(* PLC project tennessee-eastman-chemical, Generated TextualNotationConverter 1.0 *)
(* stored: creationDateTime 2025-07-30T12:00:00, modificationDateTime 2025-01-30T12:00:00 *)

FUNCTION_BLOCK ANALOG_IN
  VAR_INPUT
    Name : STRING;
    Description : STRING;
    Raw_Signal : REAL;
    PV_High : REAL;
    PV_Low : REAL;
    Scaling_Slope : REAL;
    Scaling_Offset : REAL;
    Alarm_Enable : BOOL;
  END_VAR
  VAR_OUTPUT
    PV : REAL;
    High_Alarm : BOOL;
    Low_Alarm : BOOL;
    General_Fault : BOOL;
  END_VAR

            
          
END_FUNCTION_BLOCK

FUNCTION_BLOCK BOOL_IN
  VAR_INPUT
    Name : STRING;
    Description : STRING;
    Bool_In : BOOL;
    Alarm_OnTrue : BOOL;
    Alarm_OnFalse : BOOL;
    Latch_Enable : BOOL;
    Reset_Latch : BOOL;
  END_VAR
  VAR_OUTPUT
    Bool_Out : BOOL;
    Alarm_Active : BOOL;
    Latched_Status : BOOL;
  END_VAR

            
          
END_FUNCTION_BLOCK

FUNCTION_BLOCK DIGITAL_IN
  VAR_INPUT
    Name : STRING;
    Description : STRING;
    DI_Raw : BOOL;
    DebounceTime : STRING;
    EnableAlarm : BOOL;
  END_VAR
  VAR_OUTPUT
    DI_Out : BOOL;
    Fault_State : BOOL;
  END_VAR

            
          
END_FUNCTION_BLOCK

FUNCTION_BLOCK PID_BASIC
  VAR_INPUT
    Name : STRING;
    Description : STRING;
    AUTO : BOOL;
    PV : REAL;
    SP : REAL;
    MV_MIN : REAL;
    MV_MAX : REAL;
    X0 : REAL;
    KP : REAL;
    TR : REAL;
    TD : REAL;
    PV_High : REAL;
    PV_Low : REAL;
    Deviation_Limit : REAL;
    Inhibit : BOOL;
  END_VAR
  VAR_OUTPUT
    PV_High_Alarm : BOOL;
    PV_Low_Alarm : BOOL;
    Deviation_Alarm : BOOL;
    XOUT : REAL;
  END_VAR

            
          
END_FUNCTION_BLOCK

FUNCTION_BLOCK VALVE_ELECTRIC
  VAR_INPUT
    Name : STRING;
    Description : STRING;
    Control_Signal : REAL;
    Manual_Mode : BOOL;
    Manual_Position : REAL;
    Open_Limit : REAL;
    Close_Limit : REAL;
    Timeout : STRING;
    Inhibit : BOOL;
  END_VAR
  VAR_OUTPUT
    Valve_Position : REAL;
    Feedback_Pos : REAL;
    Valve_Moving : BOOL;
    Position_Error : BOOL;
    Alarm : BOOL;
  END_VAR

            
          
END_FUNCTION_BLOCK

FUNCTION_BLOCK VALVE_ON_OFF
  VAR_INPUT
    Name : STRING;
    Description : STRING;
    Open_Cmd : BOOL;
    Close_Cmd : BOOL;
    Timeout : STRING;
    Inhibit : BOOL;
  END_VAR
  VAR_OUTPUT
    FB_Opened : BOOL;
    FB_Closed : BOOL;
    Valve_Open_Out : BOOL;
    Valve_Close_Out : BOOL;
    Alarm_Position_Error : BOOL;
    Alarm_General : BOOL;
  END_VAR

            
          
END_FUNCTION_BLOCK

PROGRAM Section2
  VAR
    FIT_101_Raw_mA : REAL;
    FIT_101_FlowRate_GPM : REAL;
    FIC_104_MV_Percent : REAL;
    PV_103_Feedback_Position_Percent : REAL;
    PI_001_Raw_mA : REAL;
    PI_001_Pressure_psig : REAL;
  END_VAR
  VAR
    FIT-101 : ANALOG_IN;
    FIC-104 : PID_BASIC;
    PV-103 : VALVE_ELECTRIC;
    XV-106 : VALVE_ON_OFF;
    PI-001 : ANALOG_IN;
    IAL-101 : BOOL_IN;
    FAL-101 : DIGITAL_IN;
    FAL-102 : DIGITAL_IN;
    FAL-103 : DIGITAL_IN;
  END_VAR
  VAR  (* added by the conversion: wires and edge detectors of the diagram *)
    _OR2_OUT : BOOL;
  END_VAR

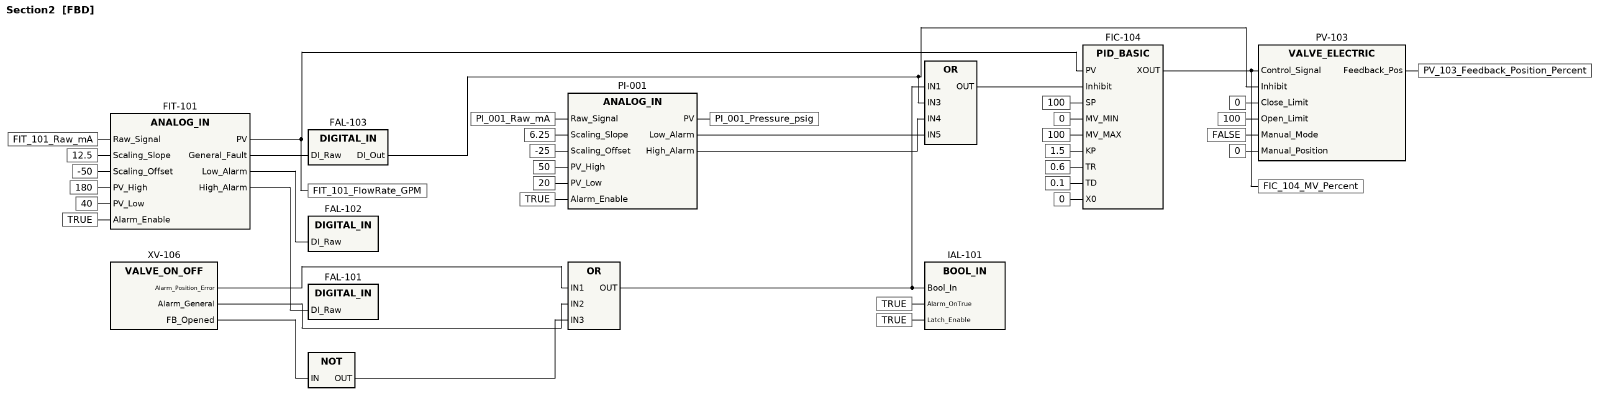
(* FBD diagram, written out as Structured Text *)
FIT-101(Raw_Signal := FIT_101_Raw_mA, Scaling_Slope := 12.5, Scaling_Offset := -50, PV_High := 180, PV_Low := 40, Alarm_Enable := TRUE);
XV-106();
_OR2_OUT := XV-106.Alarm_Position_Error OR XV-106.Alarm_General OR NOT XV-106.FB_Opened;
FAL-103(DI_Raw := FIT-101.General_Fault);
PI-001(Raw_Signal := PI_001_Raw_mA, Scaling_Slope := 6.25, Scaling_Offset := -25, PV_High := 50, PV_Low := 20, Alarm_Enable := TRUE);
FIC-104(PV := FIT-101.PV, Inhibit := _OR2_OUT OR FAL-103.DI_Out OR PI-001.High_Alarm OR PI-001.Low_Alarm, SP := 100, MV_MIN := 0, MV_MAX := 100, KP := 1.5, TR := 0.6, TD := 0.1, X0 := 0);
FIC_104_MV_Percent := FIC-104.XOUT;
FIT_101_FlowRate_GPM := FIT-101.PV;
PI_001_Pressure_psig := PI-001.PV;
PV-103(Control_Signal := FIC-104.XOUT, Inhibit := FAL-103.DI_Out, Close_Limit := 0, Open_Limit := 100, Manual_Mode := FALSE, Manual_Position := 0);
PV_103_Feedback_Position_Percent := PV-103.Feedback_Pos;
IAL-101(Bool_In := _OR2_OUT, Alarm_OnTrue := TRUE, Latch_Enable := TRUE);
FAL-101(DI_Raw := FIT-101.High_Alarm);
FAL-102(DI_Raw := FIT-101.Low_Alarm);
END_PROGRAM

FUNCTION_BLOCK DUTY_STANDBY
  VAR_INPUT
    Name : STRING;
    Description : STRING;
    Enable : BOOL;
    StartRequest : BOOL;
    AlternateEnable : BOOL;
    ForcePumpA : BOOL;
    ForcePumpB : BOOL;
    DutyElapsed : BOOL;
    MinRunElapsed : BOOL;
    SwitchoverDelayElapsed : BOOL;
    StartTimeoutElapsed : BOOL;
    PumpA_RunFB : BOOL;
    PumpB_RunFB : BOOL;
    PumpA_Fault : BOOL;
    PumpB_Fault : BOOL;
    Reset : BOOL;
    Inhibit : BOOL;
  END_VAR
  VAR_OUTPUT
    CmdPumpA : BOOL;
    CmdPumpB : BOOL;
    ActiveIsA : BOOL;
    SwitchedDueToDuty : BOOL;
    SwitchedDueToFailure : BOOL;
    Alarm_FailedStart_A : BOOL;
    Alarm_FailedStart_B : BOOL;
    Alarm_NoAvailablePump : BOOL;
  END_VAR

            
          
END_FUNCTION_BLOCK

FUNCTION_BLOCK MOTOR_2SPD
  VAR_INPUT
    Name : STRING;
    Description : STRING;
    Start_Cmd : BOOL;
    Stop_Cmd : BOOL;
    Speed_High_Cmd : BOOL;
    Speed_Low_Cmd : BOOL;
    Inhibit : BOOL;
  END_VAR
  VAR_OUTPUT
    Motor_Start_Out : BOOL;
    FB_Running : BOOL;
    FB_Trip : BOOL;
    FB_HighSpeed : BOOL;
    FB_LowSpeed : BOOL;
    Alarm_Speed_Error : BOOL;
  END_VAR

            
          
END_FUNCTION_BLOCK

FUNCTION_BLOCK MOTOR_ON_OFF
  VAR_INPUT
    Name : STRING;
    Description : STRING;
    Start_Cmd : BOOL;
    Stop_Cmd : BOOL;
    Start_Delay : STRING;
    MinRunTime : STRING;
    Inhibit : BOOL;
  END_VAR
  VAR_OUTPUT
    Motor_Start_Out : BOOL;
    FB_Running : BOOL;
    FB_Trip : BOOL;
    Alarm_Start_Fail : BOOL;
    Alarm_Stop_Fail : BOOL;
  END_VAR

            
          
END_FUNCTION_BLOCK

FUNCTION_BLOCK MOTOR_VSD
  VAR_INPUT
    Name : STRING;
    Description : STRING;
    Start_Cmd : BOOL;
    Stop_Cmd : BOOL;
    Speed_SP : REAL;
    Accel_Ramp : STRING;
    Decel_Ramp : STRING;
    Inhibit : BOOL;
  END_VAR
  VAR_OUTPUT
    Speed_Out : REAL;
    FB_Running : BOOL;
    FB_Fault : BOOL;
    FB_Ready : BOOL;
    FB_ActualSpeed : REAL;
    Alarm_Speed_Deviation : BOOL;
    Alarm_Comm_Fail : BOOL;
  END_VAR

            
          
END_FUNCTION_BLOCK

FUNCTION_BLOCK RATIO_CONTROL
  VAR_INPUT
    Name : STRING;
    Description : STRING;
    Auto : BOOL;
    PrimaryPV : REAL;
    SecondaryPV : REAL;
    RatioSP : REAL;
    Bias : REAL;
    TrimKp : REAL;
    TrimTi : STRING;
    MV_MIN : REAL;
    MV_MAX : REAL;
    ManOut : REAL;
    Inhibit : BOOL;
  END_VAR
  VAR_OUTPUT
    SlaveSP : REAL;
    ActiveRatio : REAL;
    RatioErr : REAL;
  END_VAR

            
          
END_FUNCTION_BLOCK

FUNCTION_BLOCK SPLIT_RANGE
  VAR_INPUT
    Name : STRING;
    Description : STRING;
    IN : REAL;
    Split_Point : REAL;
    Output1_Start : REAL;
    Output1_End : REAL;
    Output2_Start : REAL;
    Output2_End : REAL;
  END_VAR
  VAR_OUTPUT
    OUT1 : REAL;
    OUT2 : REAL;
  END_VAR

            
          
END_FUNCTION_BLOCK

FUNCTION_BLOCK VOTING_ANALOG
  VAR_INPUT
    Name : STRING;
    Description : STRING;
    Input1 : REAL;
    Input2 : REAL;
    Input3 : REAL;
    Deviation_Limit : REAL;
    Voting_Scheme : STRING;
    EnableAlarm : BOOL;
    Inhibit : BOOL;
  END_VAR
  VAR_OUTPUT
    Voted_Output : REAL;
    Sensor1_Fault : BOOL;
    Sensor2_Fault : BOOL;
    Sensor3_Fault : BOOL;
    Alarm_Voting_Error : BOOL;
    Healthy_Sensors_Count : INT;
  END_VAR

            
          
END_FUNCTION_BLOCK

PROGRAM Section3
  VAR
    TIT103_PV_Temperature : REAL;
    LT105_Level_PV : REAL;
    TIC101_MV_to_XV102 : REAL;
    LIC106_MV_to_LV104 : REAL;
  END_VAR
  VAR
    TIT-103 : ANALOG_IN;
    LT-105 : ANALOG_IN;
    FC-004 : ANALOG_IN;
    TIC-101 : PID_BASIC;
    LIC-106 : PID_BASIC;
    XV-102 : VALVE_ELECTRIC;
    LV-104 : VALVE_ELECTRIC;
  END_VAR

(* FBD diagram, written out as Structured Text *)
LT-105(PV_High := 80.0, PV_Low := 20.0, Alarm_Enable := TRUE, Scaling_Slope := 6.25, Scaling_Offset := -25.0);
LV-104(Control_Signal := LIC-106.XOUT, Inhibit := LT-105.High_Alarm, Manual_Mode := LT-105.High_Alarm, Open_Limit := 100.0, Close_Limit := 0.0, Manual_Position := 0.0);
TIT-103(PV_High := 200.0, PV_Low := 160.0, Alarm_Enable := TRUE, Scaling_Slope := 15.625, Scaling_Offset := -62.5);
FC-004(PV_Low := 10.0, Alarm_Enable := TRUE);
TIC-101(PV := TIT-103.PV, Inhibit := XV-102.Position_Error OR TIT-103.High_Alarm OR FC-004.Low_Alarm OR TIT-103.General_Fault, AUTO := TON(FC-004.PV > 10.0, T#21s) AND NOT XV-102.Position_Error, SP := 180.0, MV_MIN := 0.0, MV_MAX := 100.0, KP := 3.0, TR := 1.2, TD := 0.1, PV_High := 200.0, PV_Low := 160.0);
XV-102(Control_Signal := TIC-101.XOUT, Inhibit := TIT-103.High_Alarm, Manual_Mode := TIT-103.High_Alarm, Open_Limit := 100.0, Close_Limit := 0.0, Timeout := T#5s, Manual_Position := 0.0);
LIC-106(PV := LT-105.PV, Inhibit := LV-104.Position_Error OR LT-105.General_Fault OR XV-102.Alarm, AUTO := NOT XV-102.Alarm AND TON(TIC-101.AUTO, T#15s) AND NOT LV-104.Position_Error, SP := 50.0, MV_MIN := 0.0, MV_MAX := 100.0, KP := 2.5, TR := 0.9, TD := 0.0, PV_High := 80.0, PV_Low := 20.0);
LIC106_MV_to_LV104 := LIC-106.XOUT;
LT105_Level_PV := LT-105.PV;
TIC101_MV_to_XV102 := TIC-101.XOUT;
TIT103_PV_Temperature := TIT-103.PV;
END_PROGRAM

PROGRAM Section4
  VAR
    LAH-101 : BOOL;
    LAL-101 : BOOL;
    FTL-101 : BOOL;
    LT104_Level_PV_Percent : REAL;
    LIC101_CO_PV102_CMD : REAL;
  END_VAR
  VAR
    LT-104 : ANALOG_IN;
    FIT-103 : ANALOG_IN;
    LIC-101 : PID_BASIC;
    PV-102 : VALVE_ELECTRIC;
  END_VAR

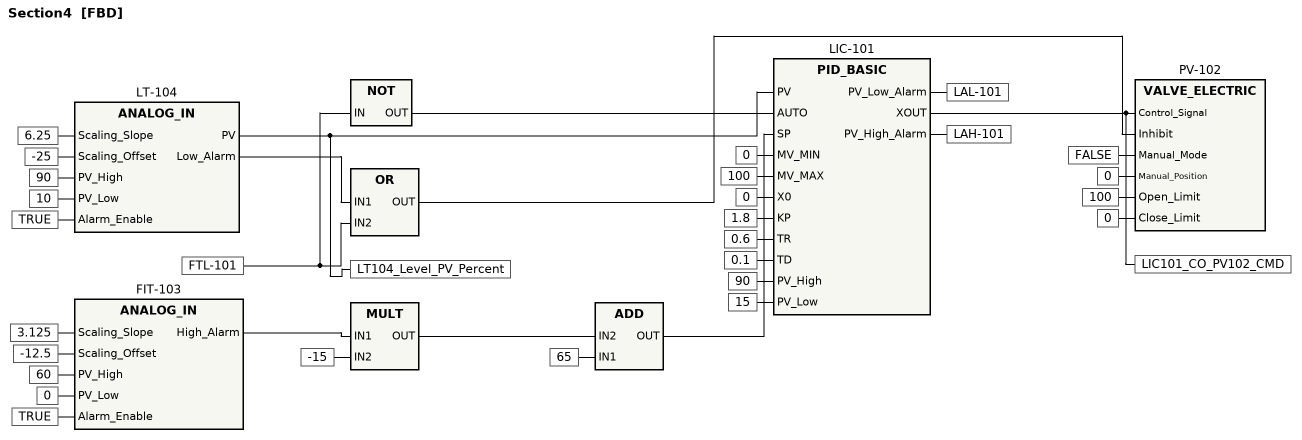
(* FBD diagram, written out as Structured Text *)
LT-104(Scaling_Slope := 6.25, Scaling_Offset := -25, PV_High := 90, PV_Low := 10, Alarm_Enable := TRUE);
FIT-103(Scaling_Slope := 3.125, Scaling_Offset := -12.5, PV_High := 60, PV_Low := 0, Alarm_Enable := TRUE);
LIC-101(PV := LT-104.PV, AUTO := NOT (FTL-101), SP := MULT(FIT-103.High_Alarm, -15) + 65, MV_MIN := 0, MV_MAX := 100, X0 := 0, KP := 1.8, TR := 0.6, TD := 0.1, PV_High := 90, PV_Low := 15);
LAH-101 := LIC-101.PV_High_Alarm;
LAL-101 := LIC-101.PV_Low_Alarm;
LIC101_CO_PV102_CMD := LIC-101.XOUT;
LT104_Level_PV_Percent := LT-104.PV;
PV-102(Control_Signal := LIC-101.XOUT, Inhibit := LT-104.Low_Alarm OR (FTL-101), Manual_Mode := FALSE, Manual_Position := 0, Open_Limit := 100, Close_Limit := 0);
END_PROGRAM

PROGRAM Section5
  VAR
    TIT106_TemperaturePV : REAL;
    TIC106_SteamFlowMV : REAL;
    FV105_SteamValvePosition : REAL;
    LT107_ColumnLevelPV : REAL;
    LIC107_LevelControlMV : REAL;
    LV102_LevelValvePosition : REAL;
    TIT106_RawSignal_mA : REAL;
    LT107_RawSignal_mA : REAL;
    CondReturn_LS_Raw : BOOL;
    COND_RETURN_OPEN_DebounceTime : TIME;
    COND_RETURN_OPEN_EnableAlarm : BOOL;
    LIC107_Manual_Request : BOOL;
  END_VAR
  VAR
    TIT-106 : ANALOG_IN;
    TIC-106 : PID_BASIC;
    FV-105 : VALVE_ELECTRIC;
    LT-107 : ANALOG_IN;
    LIC-107 : PID_BASIC;
    LV-102 : VALVE_ELECTRIC;
    COND-RETURN-OPEN-LS : DIGITAL_IN;
    FV-105-PERM-CONDR-OPEN : BOOL_IN;
    LV-102-LOWLEVEL-INTERLOCK : BOOL_IN;
    FV-105-HIGHTEMP-INTERLOCK : BOOL_IN;
  END_VAR

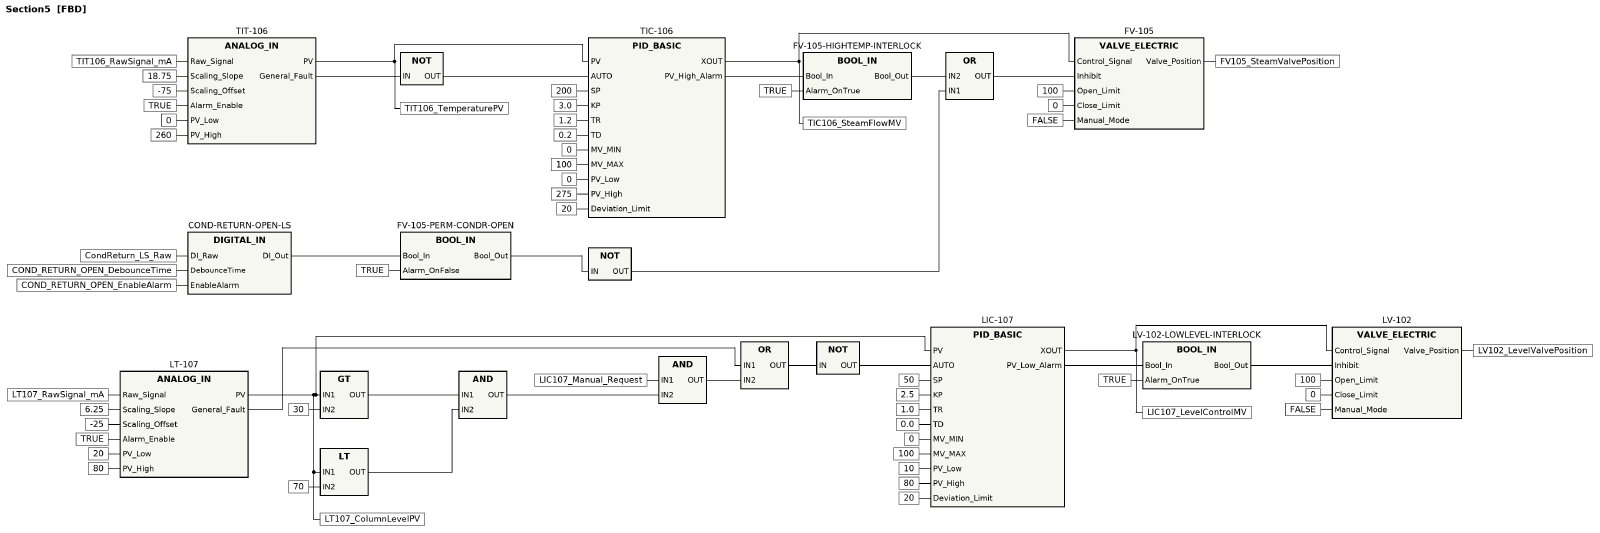
(* FBD diagram, written out as Structured Text *)
TIT-106(Raw_Signal := TIT106_RawSignal_mA, Scaling_Slope := 18.75, Scaling_Offset := -75, Alarm_Enable := TRUE, PV_Low := 0, PV_High := 260);
TIC-106(PV := TIT-106.PV, AUTO := NOT TIT-106.General_Fault, SP := 200, KP := 3.0, TR := 1.2, TD := 0.2, MV_MIN := 0, MV_MAX := 100, PV_Low := 0, PV_High := 275, Deviation_Limit := 20);
FV-105-HIGHTEMP-INTERLOCK(Bool_In := TIC-106.PV_High_Alarm, Alarm_OnTrue := TRUE);
COND-RETURN-OPEN-LS(DI_Raw := CondReturn_LS_Raw, DebounceTime := COND_RETURN_OPEN_DebounceTime, EnableAlarm := COND_RETURN_OPEN_EnableAlarm);
FV-105-PERM-CONDR-OPEN(Bool_In := COND-RETURN-OPEN-LS.DI_Out, Alarm_OnFalse := TRUE);
FV-105(Control_Signal := TIC-106.XOUT, Inhibit := FV-105-HIGHTEMP-INTERLOCK.Bool_Out OR NOT FV-105-PERM-CONDR-OPEN.Bool_Out, Open_Limit := 100, Close_Limit := 0, Manual_Mode := FALSE);
FV105_SteamValvePosition := FV-105.Valve_Position;
LT-107(Raw_Signal := LT107_RawSignal_mA, Scaling_Slope := 6.25, Scaling_Offset := -25, Alarm_Enable := TRUE, PV_Low := 20, PV_High := 80);
LIC-107(PV := LT-107.PV, AUTO := NOT (LT-107.General_Fault OR LIC107_Manual_Request AND LT-107.PV > 30 AND LT-107.PV < 70), SP := 50, KP := 2.5, TR := 1.0, TD := 0.0, MV_MIN := 0, MV_MAX := 100, PV_Low := 10, PV_High := 80, Deviation_Limit := 20);
LIC107_LevelControlMV := LIC-107.XOUT;
LT107_ColumnLevelPV := LT-107.PV;
LV-102-LOWLEVEL-INTERLOCK(Bool_In := LIC-107.PV_Low_Alarm, Alarm_OnTrue := TRUE);
LV-102(Control_Signal := LIC-107.XOUT, Inhibit := LV-102-LOWLEVEL-INTERLOCK.Bool_Out, Open_Limit := 100, Close_Limit := 0, Manual_Mode := FALSE);
LV102_LevelValvePosition := LV-102.Valve_Position;
TIC106_SteamFlowMV := TIC-106.XOUT;
TIT106_TemperaturePV := TIT-106.PV;
END_PROGRAM

PROGRAM Section6
  VAR
    TIC101_MV_To_FV103 : REAL;
    PIC501_MV_To_VentValve : REAL;
    LIC102_MV_To_FC006 : REAL;
  END_VAR
  VAR
    TI-006 : ANALOG_IN;
    TIC-101 : PID_BASIC;
    FV-103 : VALVE_ELECTRIC;
    PIT-104 : ANALOG_IN;
    PIC-501 : PID_BASIC;
    LT-102 : ANALOG_IN;
    LIC-102 : PID_BASIC;
    FC-006 : VALVE_ELECTRIC;
  END_VAR

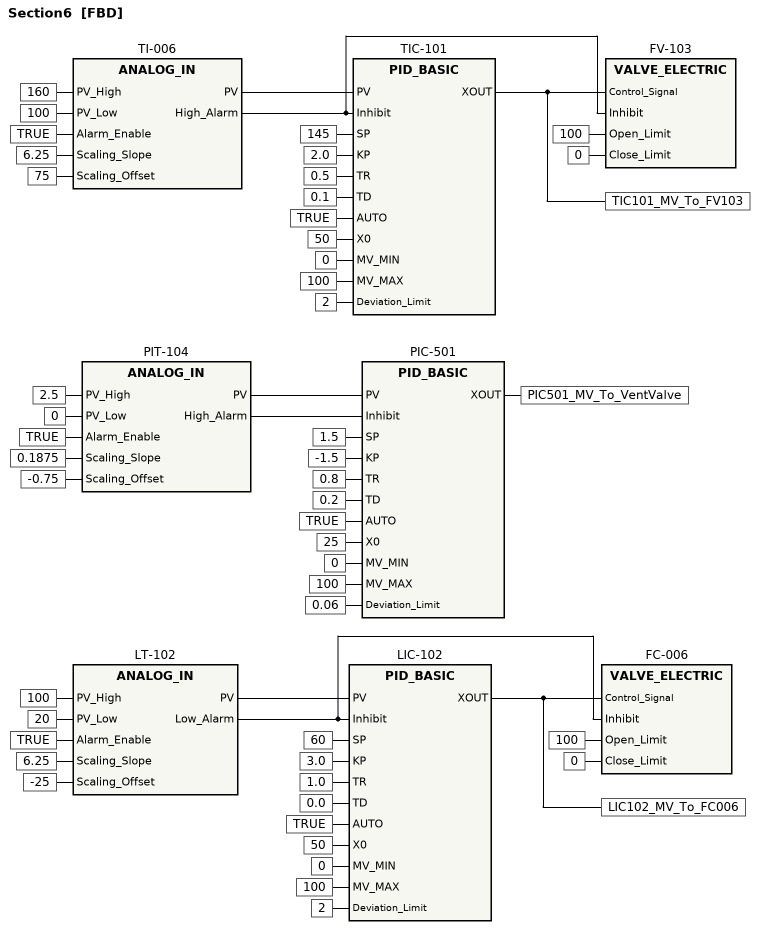
(* FBD diagram, written out as Structured Text *)
LT-102(PV_High := 100, PV_Low := 20, Alarm_Enable := TRUE, Scaling_Slope := 6.25, Scaling_Offset := -25);
LIC-102(PV := LT-102.PV, Inhibit := LT-102.Low_Alarm, SP := 60, KP := 3.0, TR := 1.0, TD := 0.0, AUTO := TRUE, X0 := 50, MV_MIN := 0, MV_MAX := 100, Deviation_Limit := 2);
LIC102_MV_To_FC006 := LIC-102.XOUT;
PIT-104(PV_High := 2.5, PV_Low := 0, Alarm_Enable := TRUE, Scaling_Slope := 0.1875, Scaling_Offset := -0.75);
PIC-501(PV := PIT-104.PV, Inhibit := PIT-104.High_Alarm, SP := 1.5, KP := -1.5, TR := 0.8, TD := 0.2, AUTO := TRUE, X0 := 25, MV_MIN := 0, MV_MAX := 100, Deviation_Limit := 0.06);
PIC501_MV_To_VentValve := PIC-501.XOUT;
TI-006(PV_High := 160, PV_Low := 100, Alarm_Enable := TRUE, Scaling_Slope := 6.25, Scaling_Offset := 75);
TIC-101(PV := TI-006.PV, Inhibit := TI-006.High_Alarm, SP := 145, KP := 2.0, TR := 0.5, TD := 0.1, AUTO := TRUE, X0 := 50, MV_MIN := 0, MV_MAX := 100, Deviation_Limit := 2);
TIC101_MV_To_FV103 := TIC-101.XOUT;
FV-103(Control_Signal := TIC-101.XOUT, Inhibit := TI-006.High_Alarm, Open_Limit := 100, Close_Limit := 0);
FC-006(Control_Signal := LIC-102.XOUT, Inhibit := LT-102.Low_Alarm, Open_Limit := 100, Close_Limit := 0);
END_PROGRAM

PROGRAM Section7
  VAR
    TIC106_SteamValveCmd_Pct : REAL;
    LIC103_OutflowValveCmd_Pct : REAL;
    LIC101_CondensateLevel_Pct : REAL;
    StartCmd : BOOL;
  END_VAR
  VAR
    LI-003 : ANALOG_IN;
    TI-008 : ANALOG_IN;
    LIC-101 : PID_BASIC;
    LIC-103 : PID_BASIC;
    TIC-106 : PID_BASIC;
    XV-104 : VALVE_ELECTRIC;
    XV-105 : VALVE_ELECTRIC;
    StartDelay : TON;
  END_VAR
  VAR  (* added by the conversion: wires and edge detectors of the diagram *)
    _OR268_OUT : BOOL;
    _NOT273_OUT : BOOL;
  END_VAR

(* FBD diagram, written out as Structured Text *)
LI-003(Scaling_Slope := 6.25, Scaling_Offset := -25, PV_Low := 10, Alarm_Enable := TRUE);
_OR268_OUT := LI-003.Low_Alarm OR LI-003.General_Fault;
LIC-103(PV := LI-003.PV, Inhibit := _OR268_OUT, SP := 70, KP := 2.5, TR := 0.8, TD := 0.1, MV_MIN := 0, MV_MAX := 100, AUTO := TRUE, PV_Low := 15);
LIC103_OutflowValveCmd_Pct := LIC-103.XOUT;
TI-008(PV_High := 195, Scaling_Slope := 15.625, Scaling_Offset := -62.5, Alarm_Enable := TRUE);
LIC-101(PV := LIC101_CondensateLevel_Pct, PV_High := 85);
StartDelay(IN := StartCmd, PT := T#12s);
_NOT273_OUT := NOT (LI-003.PV > 30 AND StartDelay.Q);
TIC-106(PV := TI-008.PV, Inhibit := LIC-101.PV_High_Alarm OR TI-008.General_Fault OR TIC-106.PV_High_Alarm OR _NOT273_OUT, AUTO := NOT LIC-101.PV_High_Alarm, SP := 180, KP := 3.2, TR := 1.0, TD := 0.3, MV_MIN := 5, MV_MAX := 95, Deviation_Limit := 10, PV_High := 210);
TIC106_SteamValveCmd_Pct := TIC-106.XOUT;
XV-104(Control_Signal := LIC-103.XOUT, Inhibit := LIC-103.PV_Low_Alarm OR _OR268_OUT, Open_Limit := 100, Close_Limit := 0);
XV-105(Control_Signal := TIC-106.XOUT, Inhibit := TI-008.General_Fault OR TIC-106.PV_High_Alarm OR LIC-101.PV_High_Alarm OR TI-008.PV > 200 OR _NOT273_OUT, Manual_Mode := TI-008.PV > 210, Open_Limit := 100, Close_Limit := 0, Manual_Position := 0);
END_PROGRAM

PROGRAM Section8
  VAR
    System_RunCmd : BOOL;
    Decanter2_Online : BOOL;
    LIC106_MV_XV101_Command : REAL;
    FC008_MV_PV104_Command : REAL;
  END_VAR
  VAR
    LT-102 : ANALOG_IN;
    LT-103 : ANALOG_IN;
    LT-107 : ANALOG_IN;
    FIT-105 : ANALOG_IN;
    LIC-106 : PID_BASIC;
    FC-008 : PID_BASIC;
    XV-101 : VALVE_ELECTRIC;
    PV-104 : VALVE_ELECTRIC;
  END_VAR
  VAR  (* added by the conversion: wires and edge detectors of the diagram *)
    _TON338_OUT : BOOL;
    _OR330_OUT : BOOL;
  END_VAR

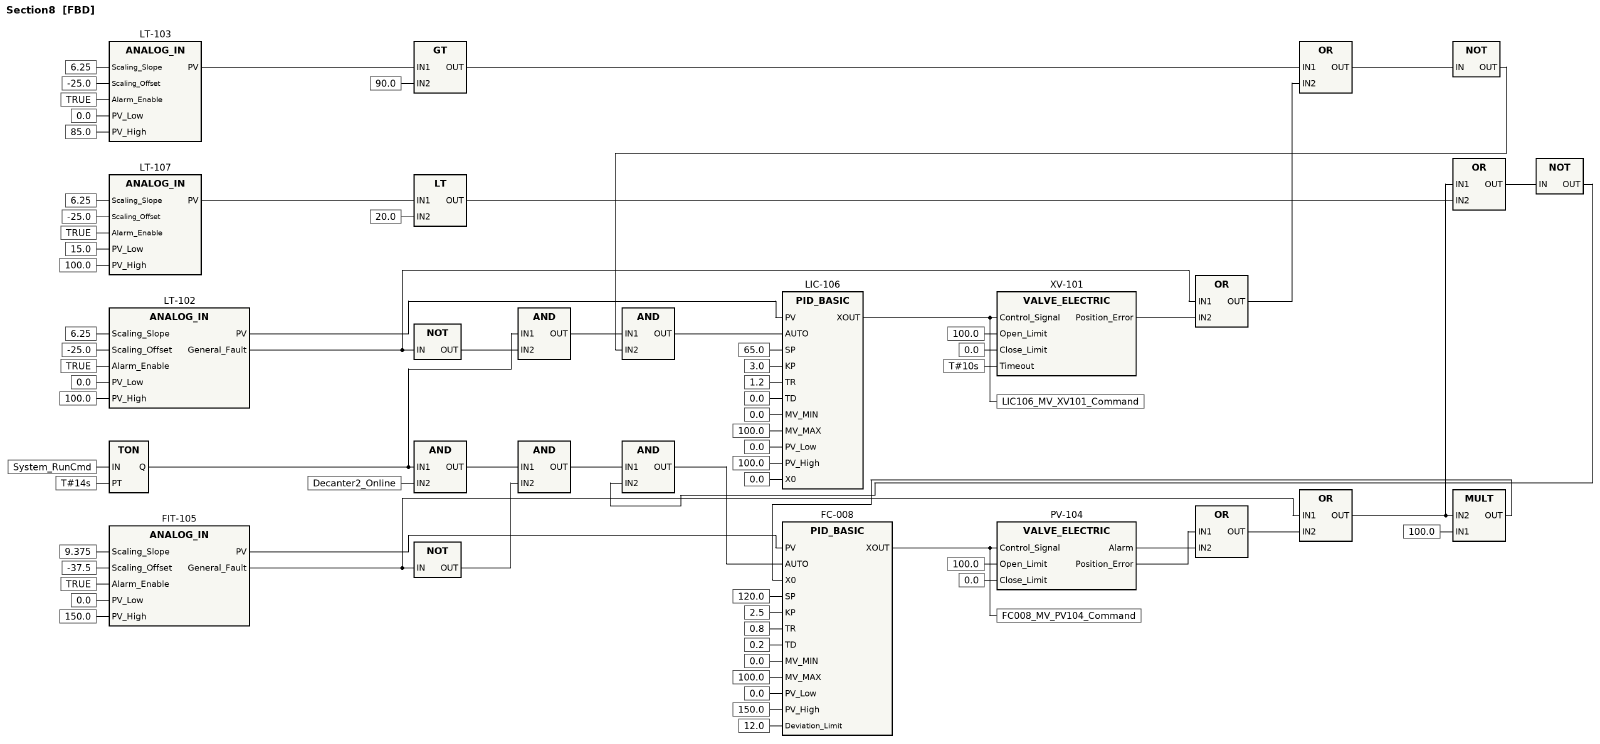
(* FBD diagram, written out as Structured Text *)
FIT-105(Scaling_Slope := 9.375, Scaling_Offset := -37.5, Alarm_Enable := TRUE, PV_Low := 0.0, PV_High := 150.0);
_TON338_OUT := TON(System_RunCmd, T#14s);
PV-104(Control_Signal := FC-008.XOUT, Open_Limit := 100.0, Close_Limit := 0.0);
_OR330_OUT := FIT-105.General_Fault OR PV-104.Position_Error OR PV-104.Alarm;
LT-107(Scaling_Slope := 6.25, Scaling_Offset := -25.0, Alarm_Enable := TRUE, PV_Low := 15.0, PV_High := 100.0);
FC-008(PV := FIT-105.PV, AUTO := _TON338_OUT AND Decanter2_Online AND NOT FIT-105.General_Fault AND NOT (_OR330_OUT OR LT-107.PV < 20.0), X0 := MULT(_OR330_OUT, 100.0), SP := 120.0, KP := 2.5, TR := 0.8, TD := 0.2, MV_MIN := 0.0, MV_MAX := 100.0, PV_Low := 0.0, PV_High := 150.0, Deviation_Limit := 12.0);
FC008_MV_PV104_Command := FC-008.XOUT;
LT-102(Scaling_Slope := 6.25, Scaling_Offset := -25.0, Alarm_Enable := TRUE, PV_Low := 0.0, PV_High := 100.0);
LT-103(Scaling_Slope := 6.25, Scaling_Offset := -25.0, Alarm_Enable := TRUE, PV_Low := 0.0, PV_High := 85.0);
XV-101(Control_Signal := LIC-106.XOUT, Open_Limit := 100.0, Close_Limit := 0.0, Timeout := T#10s);
LIC-106(PV := LT-102.PV, AUTO := _TON338_OUT AND NOT LT-102.General_Fault AND NOT (LT-103.PV > 90.0 OR LT-102.General_Fault OR XV-101.Position_Error), SP := 65.0, KP := 3.0, TR := 1.2, TD := 0.0, MV_MIN := 0.0, MV_MAX := 100.0, PV_Low := 0.0, PV_High := 100.0, X0 := 0.0);
LIC106_MV_XV101_Command := LIC-106.XOUT;
END_PROGRAM

PROGRAM Section9
  VAR
    TIT101_OverheadTempPV : REAL;
    FIC103_ControlOutputPercent : REAL;
    LV102_ValvePositionPercent : REAL;
    FI103_CoolingMediumFlowPV : REAL;
    XV104_OpenStatus : BOOL;
    LC002_ValidLevelPermissive : BOOL;
    LC002_LevelActive : BOOL;
  END_VAR
  VAR
    TIT-101 : ANALOG_IN;
    FI-103 : ANALOG_IN;
    FIC-103 : PID_BASIC;
    LV-102 : VALVE_ELECTRIC;
    XV-104 : VALVE_ON_OFF;
    XV-104_OPEN : BOOL_IN;
    LC-002_VALID : BOOL_IN;
  END_VAR
  VAR  (* added by the conversion: wires and edge detectors of the diagram *)
    _OR401_OUT : BOOL;
  END_VAR

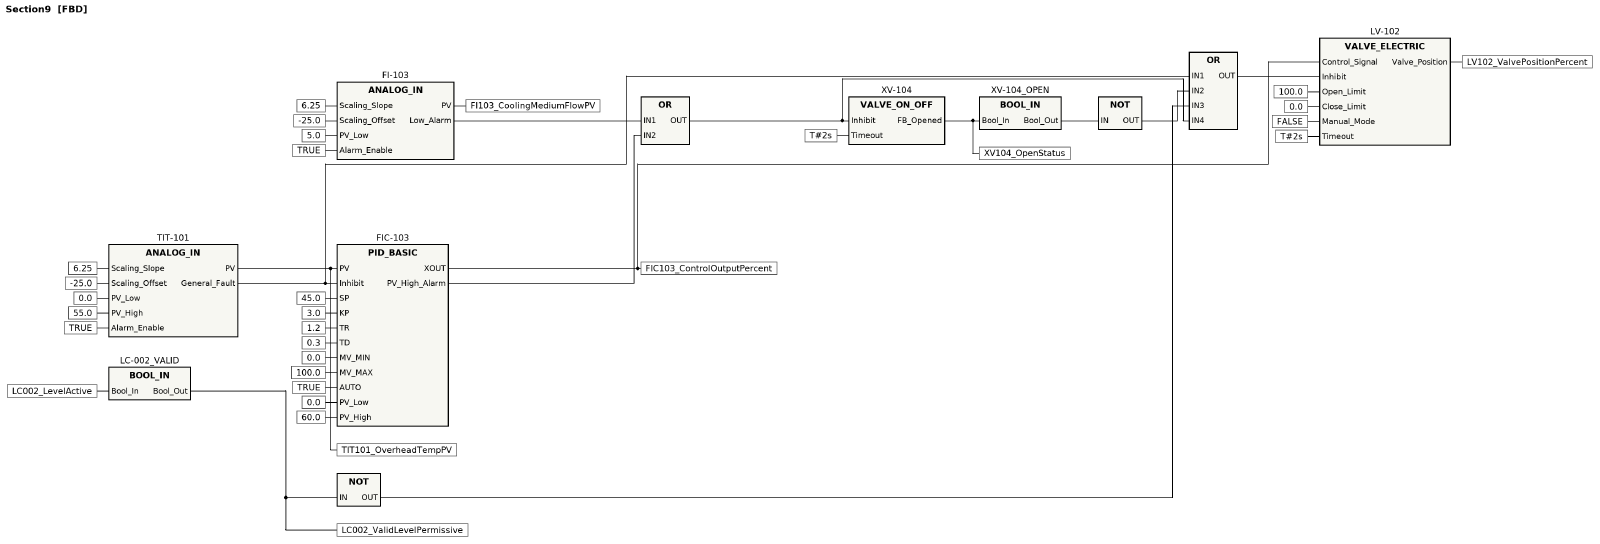
(* FBD diagram, written out as Structured Text *)
FI-103(Scaling_Slope := 6.25, Scaling_Offset := -25.0, PV_Low := 5.0, Alarm_Enable := TRUE);
FI103_CoolingMediumFlowPV := FI-103.PV;
TIT-101(Scaling_Slope := 6.25, Scaling_Offset := -25.0, PV_Low := 0.0, PV_High := 55.0, Alarm_Enable := TRUE);
FIC-103(PV := TIT-101.PV, Inhibit := TIT-101.General_Fault, SP := 45.0, KP := 3.0, TR := 1.2, TD := 0.3, MV_MIN := 0.0, MV_MAX := 100.0, AUTO := TRUE, PV_Low := 0.0, PV_High := 60.0);
FIC103_ControlOutputPercent := FIC-103.XOUT;
LC-002_VALID(Bool_In := LC002_LevelActive);
LC002_ValidLevelPermissive := LC-002_VALID.Bool_Out;
_OR401_OUT := FI-103.Low_Alarm OR FIC-103.PV_High_Alarm;
XV-104(Inhibit := _OR401_OUT, Timeout := T#2s);
XV-104_OPEN(Bool_In := XV-104.FB_Opened);
LV-102(Control_Signal := FIC-103.XOUT, Inhibit := TIT-101.General_Fault OR NOT XV-104_OPEN.Bool_Out OR NOT LC-002_VALID.Bool_Out OR _OR401_OUT, Open_Limit := 100.0, Close_Limit := 0.0, Manual_Mode := FALSE, Timeout := T#2s);
LV102_ValvePositionPercent := LV-102.Valve_Position;
TIT101_OverheadTempPV := TIT-101.PV;
XV104_OpenStatus := XV-104.FB_Opened;
END_PROGRAM

PROGRAM Section10
  VAR
    FIT_102_Raw_mA : REAL;
    LT_201_Raw_mA : REAL;
    FIT_102_Flow_PV : REAL;
    LT_201_Level_PV : REAL;
    IIC_103_CO_to_LV_101 : REAL;
    IIC_103_SP : REAL;
  END_VAR
  VAR
    FIT-102 : ANALOG_IN;
    IIC-103 : PID_BASIC;
    LV-101 : VALVE_ELECTRIC;
    LT-201 : ANALOG_IN;
    FIF-102 : BOOL_IN;
    LIH-201 : BOOL_IN;
    LC-002 : BOOL_IN;
    VAF-101 : BOOL_IN;
    FAH-102 : BOOL_IN;
    FAL-102 : BOOL_IN;
  END_VAR
  VAR  (* added by the conversion: wires and edge detectors of the diagram *)
    _OR440_OUT : BOOL;
  END_VAR

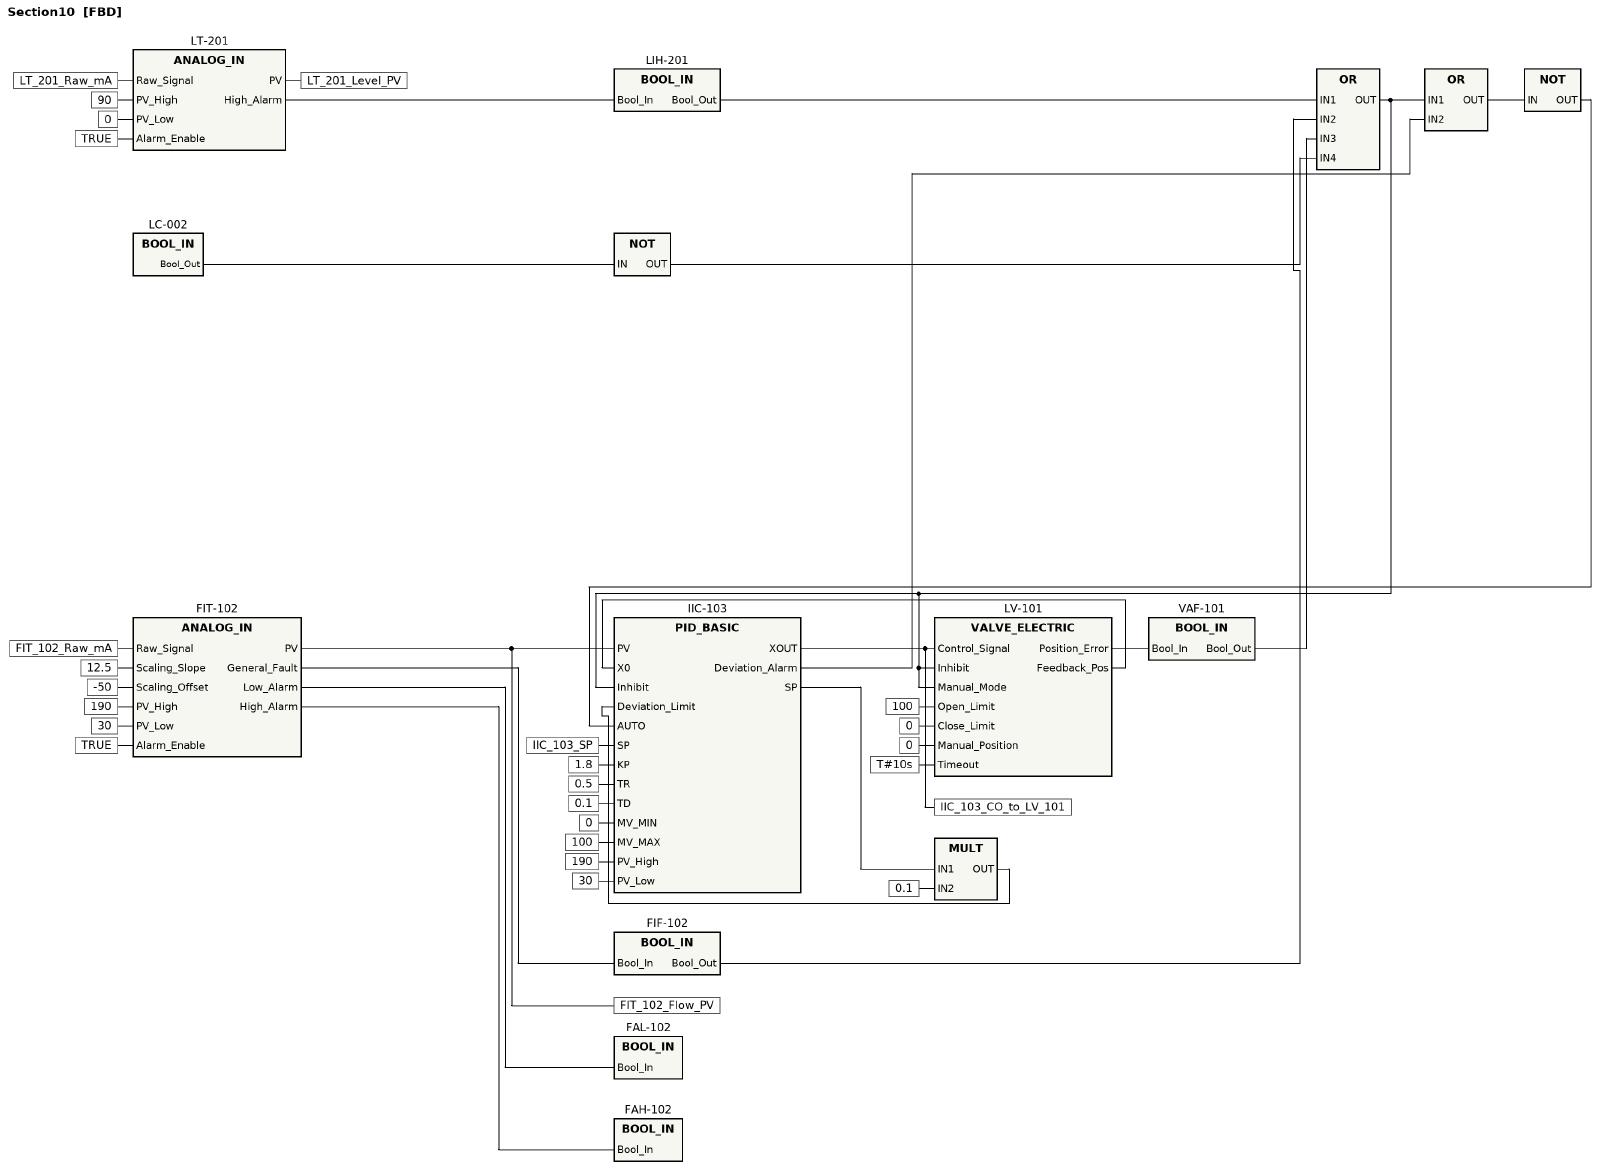
(* FBD diagram, written out as Structured Text *)
FIT-102(Raw_Signal := FIT_102_Raw_mA, Scaling_Slope := 12.5, Scaling_Offset := -50, PV_High := 190, PV_Low := 30, Alarm_Enable := TRUE);
FIT_102_Flow_PV := FIT-102.PV;
LT-201(Raw_Signal := LT_201_Raw_mA, PV_High := 90, PV_Low := 0, Alarm_Enable := TRUE);
LIH-201(Bool_In := LT-201.High_Alarm);
FIF-102(Bool_In := FIT-102.General_Fault);
VAF-101(Bool_In := LV-101.Position_Error);
LC-002();
_OR440_OUT := LIH-201.Bool_Out OR FIF-102.Bool_Out OR VAF-101.Bool_Out OR NOT LC-002.Bool_Out;
LV-101(Control_Signal := IIC-103.XOUT, Inhibit := _OR440_OUT, Manual_Mode := _OR440_OUT, Open_Limit := 100, Close_Limit := 0, Manual_Position := 0, Timeout := T#10s);
IIC-103(PV := FIT-102.PV, X0 := LV-101.Feedback_Pos, Inhibit := _OR440_OUT, Deviation_Limit := MULT(IIC-103.SP, 0.1), AUTO := NOT (_OR440_OUT OR IIC-103.Deviation_Alarm), SP := IIC_103_SP, KP := 1.8, TR := 0.5, TD := 0.1, MV_MIN := 0, MV_MAX := 100, PV_High := 190, PV_Low := 30);
IIC_103_CO_to_LV_101 := IIC-103.XOUT;
LT_201_Level_PV := LT-201.PV;
FAH-102(Bool_In := FIT-102.High_Alarm);
FAL-102(Bool_In := FIT-102.Low_Alarm);
END_PROGRAM

CONFIGURATION Config0
  RESOURCE Res0 ON PLC
    TASK task0(INTERVAL := T#20ms, PRIORITY := 0);
    PROGRAM instance0 WITH task0 : Section2;
    PROGRAM instance_1 WITH task0 : Section3;
    PROGRAM instance_2 WITH task0 : Section4;
    PROGRAM instance_3 WITH task0 : Section5;
    PROGRAM instance_4 WITH task0 : Section6;
    PROGRAM instance_5 WITH task0 : Section7;
    PROGRAM instance_6 WITH task0 : Section8;
    PROGRAM instance_7 WITH task0 : Section9;
    PROGRAM instance_8 WITH task0 : Section10;
  END_RESOURCE
END_CONFIGURATION
